ABB RAPID module: MainModule.mod

MODULE MainModule
	TASK PERS tooldata realsense:=[TRUE,[[103.923,60,1000],[1,0,0,0]],[2,[0,0,8],[1,0,0,0],0,0,0]];
	CONST robtarget p10:=[[824.16,73.96,149.20],[2.12842E-05,0.105952,0.994011,-0.0267822],[0,-1,-4,0],[9E+09,9E+09,9E+09,9E+09,9E+09,9E+09]];
	CONST robtarget p20:=[[824.16,73.97,149.20],[0.0193353,0.104177,0.972469,-0.207549],[0,-1,-4,0],[9E+09,9E+09,9E+09,9E+09,9E+09,9E+09]];
	CONST robtarget p30:=[[824.17,73.97,149.20],[0.0805655,-0.0821402,-0.981506,0.152997],[0,-1,-4,0],[9E+09,9E+09,9E+09,9E+09,9E+09,9E+09]];
	CONST robtarget p40:=[[824.17,73.97,149.20],[0.133355,-0.0575785,-0.989156,0.0217193],[0,-1,-4,0],[9E+09,9E+09,9E+09,9E+09,9E+09,9E+09]];
	CONST robtarget p50:=[[824.17,73.97,149.20],[0.120041,-0.0264481,-0.981847,-0.144458],[-1,0,-5,0],[9E+09,9E+09,9E+09,9E+09,9E+09,9E+09]];
	CONST robtarget p60:=[[824.16,73.97,149.20],[0.0354254,-0.00746045,0.982249,0.184056],[-1,0,-5,0],[9E+09,9E+09,9E+09,9E+09,9E+09,9E+09]];
	CONST robtarget p70:=[[824.16,73.98,149.20],[0.13839,-0.0317435,0.984089,0.106819],[-1,0,-5,0],[9E+09,9E+09,9E+09,9E+09,9E+09,9E+09]];
	CONST robtarget p80:=[[824.17,73.98,149.20],[0.230683,-0.0488191,0.971784,-0.00617196],[0,-1,-5,0],[9E+09,9E+09,9E+09,9E+09,9E+09,9E+09]];
	CONST robtarget p90:=[[824.10,73.95,149.18],[0.155173,-0.106368,0.962623,-0.194845],[0,-1,-4,0],[9E+09,9E+09,9E+09,9E+09,9E+09,9E+09]];
	CONST robtarget p100:=[[824.14,73.97,149.20],[0.0630606,0.143791,-0.90145,0.403405],[0,-1,-4,0],[9E+09,9E+09,9E+09,9E+09,9E+09,9E+09]];
	CONST robtarget p110:=[[824.16,73.97,149.19],[0.259063,0.219304,-0.918559,0.202589],[0,-1,-5,0],[9E+09,9E+09,9E+09,9E+09,9E+09,9E+09]];

    PROC takePicture(robtarget point)
        MoveJ point, v1000, z50, realsense;
        MoveL point, v20, fine, realsense;
        Set DO10_2;
        WaitTime \InPos, 1;
        Reset DO10_2;
    ENDPROC

	PROC main()
        takePicture p10;
        takePicture p20;
        takePicture p30;
        takePicture p40;
        takePicture p50;
        takePicture p60;
        takePicture p70;
        takePicture p80;
        takePicture p90;
        takePicture p100;
        takePicture p110;
        Set DO10_3;
        WaitTime \InPos, 1;
        Reset DO10_3;
	ENDPROC
ENDMODULE
